// TwinCAT 3 PLC project Instructions_Practice
// ProgramVersion: 3.1.4024.0
// libraries:
//   Tc2_Standard, * (Beckhoff Automation GmbH)
//   Tc2_System, * (Beckhoff Automation GmbH)
//   Tc3_Module, * (Beckhoff Automation GmbH)
// project tree:
//   / PlcTask.TcTTO
//   POUs/ FB_TankController.TcPOU, I_TankController.TcIO, MAIN.TcPOU
// real-time tasks:
//   TASK PlcTask: cycle T#10ms, priority 20, ADS port 350
//   TASK PlcTask1: cycle T#10ms, priority 22, ADS port 351
//   TASK PlcTask2: cycle T#10ms, priority 21, ADS port 352
//   TASK PlcTask3: cycle T#10ms, priority 23, ADS port 353
//   TASK PlcTask4: cycle T#10ms, priority 24, ADS port 354
//   TASK PlcTask5: cycle T#10ms, priority 25, ADS port 355

CONFIGURATION Instructions_Practice
    RESOURCE PLC ON TwinCAT3
        TASK PlcTask(INTERVAL := T#10ms, PRIORITY := 20);
        PROGRAM MAIN WITH PlcTask : MAIN;
    END_RESOURCE
END_CONFIGURATION

// ---- POUs/I_TankController.TcIO
INTERFACE I_TankController

METHOD ApplyCooling 
VAR_INPUT
END_VAR
END_METHOD

METHOD CheckSafety 
VAR_INPUT
END_VAR
END_METHOD

END_INTERFACE

// ---- POUs/MAIN.TcPOU
PROGRAM MAIN
VAR
	nNum1 : INT ;
	nResult : INT;
	nMark : INT := 34;
	sGrade : STRING;
	
	
	
END_VAR

Act_Condition();
Act_Switch();

ACTION Act_Condition:
IF nNum1 = 1 THEN
	nResult := 1;
ELSIF nNum1 = 2 THEN
	nResult := 2;
IF nNum1 = 2 THEN
	nResult := 15;
END_IF
ELSIF nNum1 = 3 THEN
	nResult := 3;
ELSIF nNum1 = 2 THEN
	nResult := 4;
ELSE
	nResult := 10;		
END_IF
END_ACTION

ACTION Act_Switch:
CASE nMark OF
	91..100 :
	sGrade := 'A';
	81..90 :
	sGrade := 'B';
	71..80 :
	sGrade := 'C';
	61..70 :
	sGrade := 'D';
	ELSE
		sGrade := 'F';
END_CASE
END_ACTION

END_PROGRAM

// ---- POUs/FB_TankController.TcPOU
FUNCTION_BLOCK FB_TankController IMPLEMENTS I_TankController

VAR_IN_OUT
	nNum : INT;
END_VAR
VAR
END_VAR

{warning 'add method implementation '}
METHOD ApplyCooling
END_METHOD

{warning 'add method implementation '}
METHOD CheckSafety
END_METHOD

END_FUNCTION_BLOCK
